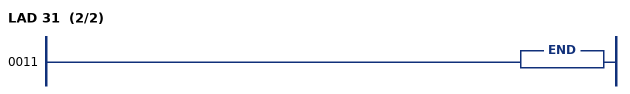
% Rung: 11 %
SOR END EOR

LADDER 32
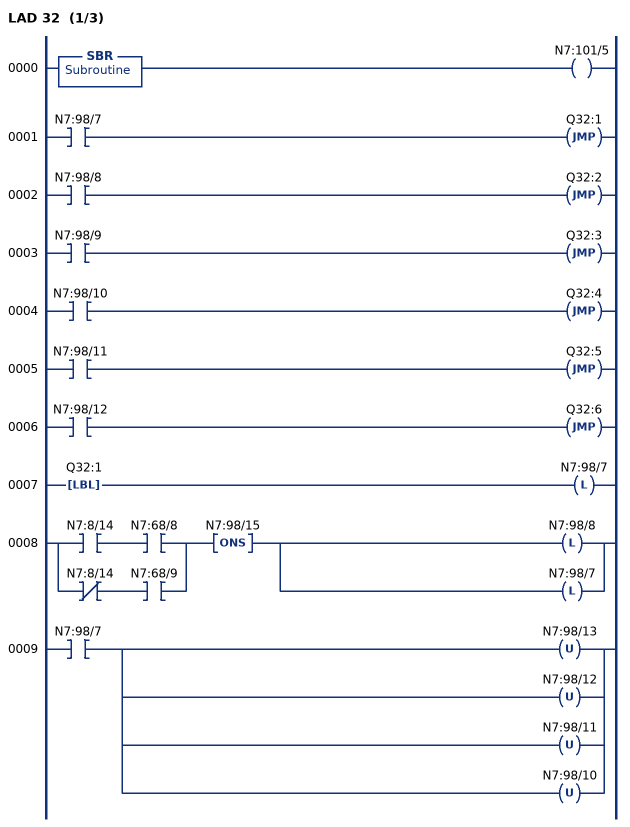
% Rung: 0 %
SOR SBR OTE N7:101/5 EOR
% Rung: 1 %
SOR XIC N7:98/7 JMP Q32:1 EOR
% Rung: 2 %
SOR XIC N7:98/8 JMP Q32:2 EOR
% Rung: 3 %
SOR XIC N7:98/9 JMP Q32:3 EOR
% Rung: 4 %
SOR XIC N7:98/10 JMP Q32:4 EOR
% Rung: 5 %
SOR XIC N7:98/11 JMP Q32:5 EOR
% Rung: 6 %
SOR XIC N7:98/12 JMP Q32:6 EOR
% Rung: 7 %
SOR LBL Q32:1 OTL N7:98/7 EOR
% Rung: 8 %
SOR BST XIC N7:8/14 XIC N7:68/8 NXB XIO N7:8/14 XIC N7:68/9 BND OSR N7:98/15 BST OTL N7:98/8 NXB OTL N7:98/7 BND EOR
% Rung: 9 %
SOR XIC N7:98/7 BST OTU N7:98/13 NXB BST OTU N7:98/12 NXB BST OTU N7:98/11 NXB OTU N7:98/10 BND BND BND EOR

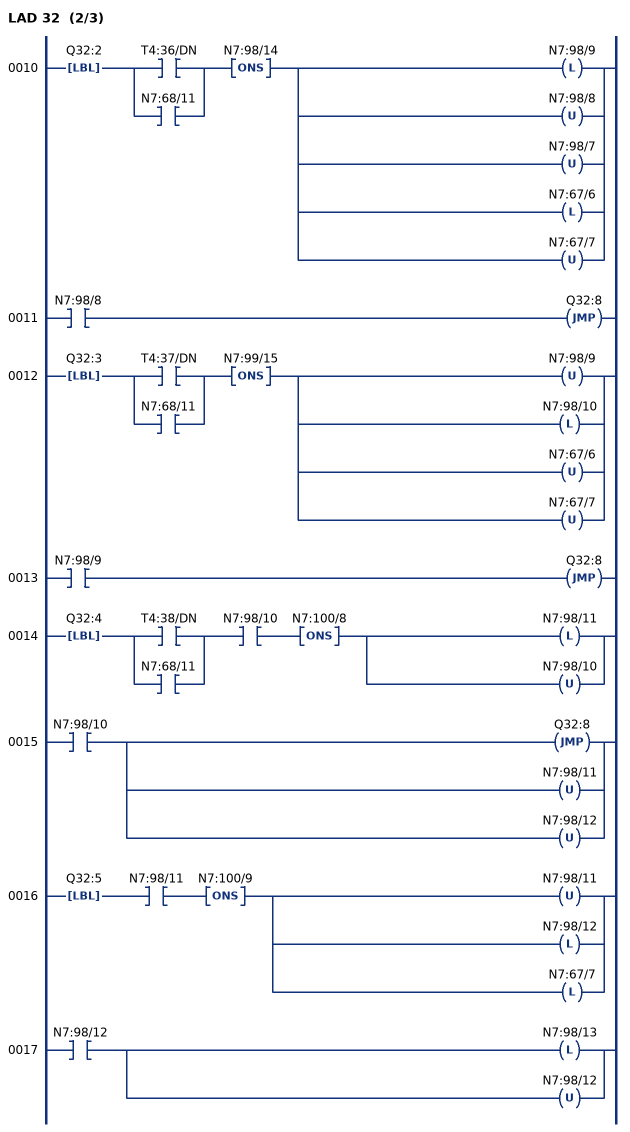
% Rung: 10 %
SOR LBL Q32:2 BST XIC T4:36/DN NXB XIC N7:68/11 BND OSR N7:98/14 BST OTL N7:98/9 NXB BST BST OTU N7:98/8 NXB OTU N7:98/7 BND NXB BST OTL N7:67/6 NXB OTU N7:67/7 BND BND BND EOR
% Rung: 11 %
SOR XIC N7:98/8 JMP Q32:8 EOR
% Rung: 12 %
SOR LBL Q32:3 BST XIC T4:37/DN NXB XIC N7:68/11 BND OSR N7:99/15 BST OTU N7:98/9 NXB BST OTL N7:98/10 NXB BST OTU N7:67/6 NXB OTU N7:67/7 BND BND BND EOR
% Rung: 13 %
SOR XIC N7:98/9 JMP Q32:8 EOR
% Rung: 14 %
SOR LBL Q32:4 BST XIC T4:38/DN NXB XIC N7:68/11 BND XIC N7:98/10 OSR N7:100/8 BST OTL N7:98/11 NXB OTU N7:98/10 BND EOR
% Rung: 15 %
SOR XIC N7:98/10 BST JMP Q32:8 NXB BST OTU N7:98/11 NXB OTU N7:98/12 BND BND EOR
% Rung: 16 %
SOR LBL Q32:5 XIC N7:98/11 OSR N7:100/9 BST BST OTU N7:98/11 NXB OTL N7:98/12 BND NXB OTL N7:67/7 BND EOR
% Rung: 17 %
SOR XIC N7:98/12 BST OTL N7:98/13 NXB OTU N7:98/12 BND EOR

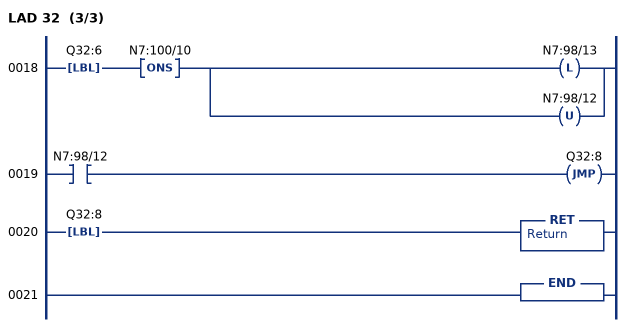
% Rung: 18 %
SOR LBL Q32:6 OSR N7:100/10 BST OTL N7:98/13 NXB OTU N7:98/12 BND EOR
% Rung: 19 %
SOR XIC N7:98/12 JMP Q32:8 EOR
% Rung: 20 %
SOR LBL Q32:8 RET EOR
% Rung: 21 %
SOR END EOR

LADDER 33
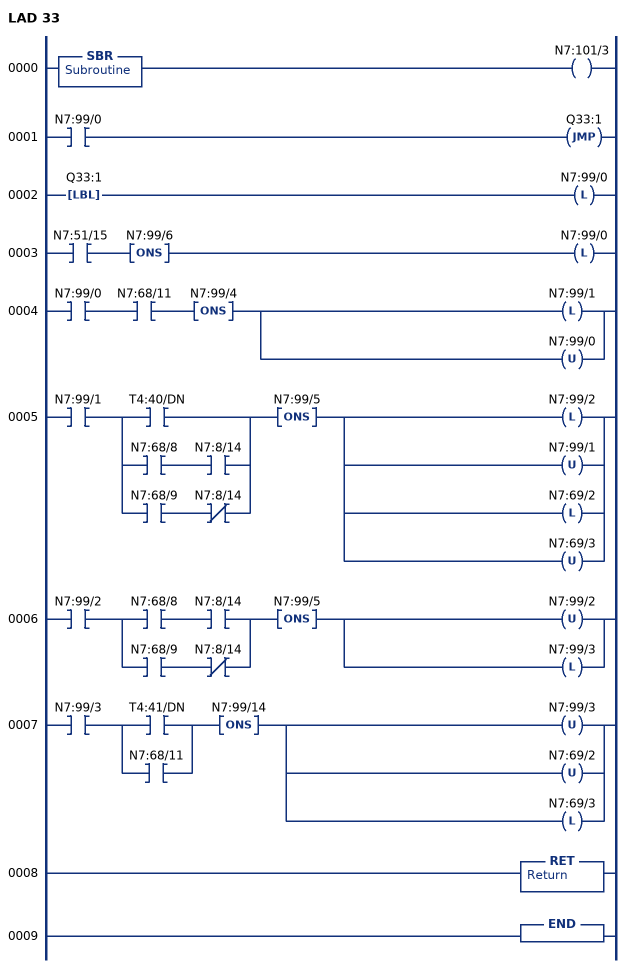
% Rung: 0 %
SOR SBR OTE N7:101/3 EOR
% Rung: 1 %
SOR XIC N7:99/0 JMP Q33:1 EOR
% Rung: 2 %
SOR LBL Q33:1 OTL N7:99/0 EOR
% Rung: 3 %
SOR XIC N7:51/15 OSR N7:99/6 OTL N7:99/0 EOR
% Rung: 4 %
SOR XIC N7:99/0 XIC N7:68/11 OSR N7:99/4 BST OTL N7:99/1 NXB OTU N7:99/0 BND EOR
% Rung: 5 %
SOR XIC N7:99/1 BST XIC T4:40/DN NXB BST XIC N7:68/8 XIC N7:8/14 NXB XIC N7:68/9 XIO N7:8/14 BND BND OSR N7:99/5 BST OTL N7:99/2 NXB BST OTU N7:99/1 NXB BST OTL N7:69/2 NXB OTU N7:69/3 BND BND BND EOR
% Rung: 6 %
SOR XIC N7:99/2 BST XIC N7:68/8 XIC N7:8/14 NXB XIC N7:68/9 XIO N7:8/14 BND OSR N7:99/5 BST OTU N7:99/2 NXB OTL N7:99/3 BND EOR
% Rung: 7 %
SOR XIC N7:99/3 BST XIC T4:41/DN NXB XIC N7:68/11 BND OSR N7:99/14 BST OTU N7:99/3 NXB BST OTU N7:69/2 NXB OTL N7:69/3 BND BND EOR
% Rung: 8 %
SOR RET EOR
% Rung: 9 %
SOR END EOR

LADDER 34
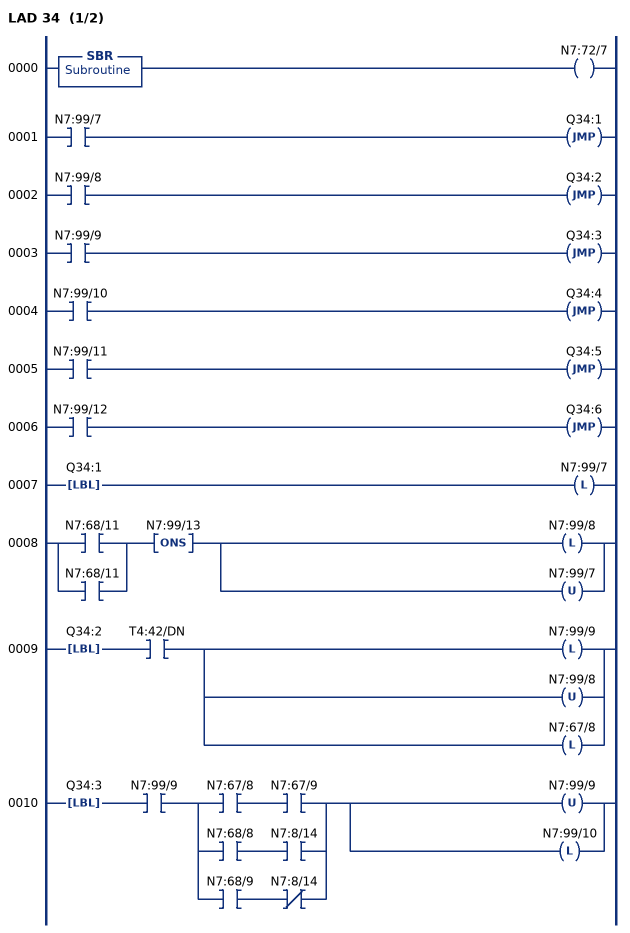
% Rung: 0 %
SOR SBR OTE N7:72/7 EOR
% Rung: 1 %
SOR XIC N7:99/7 JMP Q34:1 EOR
% Rung: 2 %
SOR XIC N7:99/8 JMP Q34:2 EOR
% Rung: 3 %
SOR XIC N7:99/9 JMP Q34:3 EOR
% Rung: 4 %
SOR XIC N7:99/10 JMP Q34:4 EOR
% Rung: 5 %
SOR XIC N7:99/11 JMP Q34:5 EOR
% Rung: 6 %
SOR XIC N7:99/12 JMP Q34:6 EOR
% Rung: 7 %
SOR LBL Q34:1 OTL N7:99/7 EOR
% Rung: 8 %
SOR BST XIC N7:68/11 NXB XIC N7:68/11 BND OSR N7:99/13 BST OTL N7:99/8 NXB OTU N7:99/7 BND EOR
% Rung: 9 %
SOR LBL Q34:2 XIC T4:42/DN BST OTL N7:99/9 NXB BST OTU N7:99/8 NXB OTL N7:67/8 BND BND EOR
% Rung: 10 %
SOR LBL Q34:3 XIC N7:99/9 BST XIC N7:67/8 XIC N7:67/9 NXB BST XIC N7:68/8 XIC N7:8/14 NXB XIC N7:68/9 XIO N7:8/14 BND BND BST OTU N7:99/9 NXB OTL N7:99/10 BND EOR

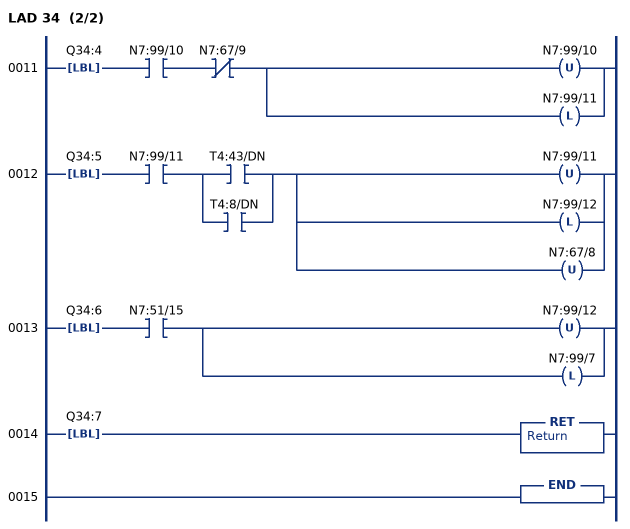
% Rung: 11 %
SOR LBL Q34:4 XIC N7:99/10 XIO N7:67/9 BST OTU N7:99/10 NXB OTL N7:99/11 BND EOR
% Rung: 12 %
SOR LBL Q34:5 XIC N7:99/11 BST XIC T4:43/DN NXB XIC T4:8/DN BND BST OTU N7:99/11 NXB BST OTL N7:99/12 NXB OTU N7:67/8 BND BND EOR
% Rung: 13 %
SOR LBL Q34:6 XIC N7:51/15 BST OTU N7:99/12 NXB OTL N7:99/7 BND EOR
% Rung: 14 %
SOR LBL Q34:7 RET EOR
% Rung: 15 %
SOR END EOR

LADDER 35
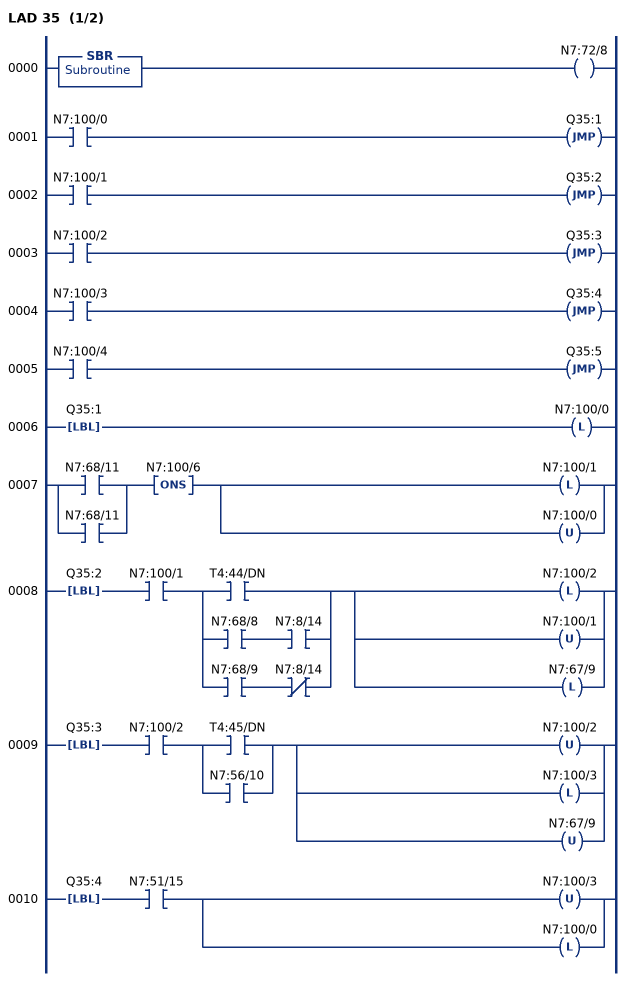
% Rung: 0 %
SOR SBR OTE N7:72/8 EOR
% Rung: 1 %
SOR XIC N7:100/0 JMP Q35:1 EOR
% Rung: 2 %
SOR XIC N7:100/1 JMP Q35:2 EOR
% Rung: 3 %
SOR XIC N7:100/2 JMP Q35:3 EOR
% Rung: 4 %
SOR XIC N7:100/3 JMP Q35:4 EOR
% Rung: 5 %
SOR XIC N7:100/4 JMP Q35:5 EOR
% Rung: 6 %
SOR LBL Q35:1 OTL N7:100/0 EOR
% Rung: 7 %
SOR BST XIC N7:68/11 NXB XIC N7:68/11 BND OSR N7:100/6 BST OTL N7:100/1 NXB OTU N7:100/0 BND EOR
% Rung: 8 %
SOR LBL Q35:2 XIC N7:100/1 BST XIC T4:44/DN NXB BST XIC N7:68/8 XIC N7:8/14 NXB XIC N7:68/9 XIO N7:8/14 BND BND BST OTL N7:100/2 NXB BST OTU N7:100/1 NXB OTL N7:67/9 BND BND EOR
% Rung: 9 %
SOR LBL Q35:3 XIC N7:100/2 BST XIC T4:45/DN NXB XIC N7:56/10 BND BST OTU N7:100/2 NXB BST OTL N7:100/3 NXB OTU N7:67/9 BND BND EOR
% Rung: 10 %
SOR LBL Q35:4 XIC N7:51/15 BST OTU N7:100/3 NXB OTL N7:100/0 BND EOR

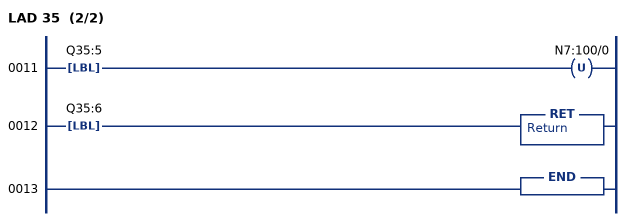
% Rung: 11 %
SOR LBL Q35:5 OTU N7:100/0 EOR
% Rung: 12 %
SOR LBL Q35:6 RET EOR
% Rung: 13 %
SOR END EOR

DATA TABLE (non-zero values as saved)
DATA T4
% .PRE .ACC %
% T4:0 % 3600 0
% T4:1 % 3800 0
% T4:2 % 3500 0
% T4:3 % 35 0
% T4:4 % 1000 0
% T4:5 % 118 0
% T4:6 % 60 0
% T4:7 % 3050 0
% T4:8 % 680 0
% T4:9 % 80 0
% T4:10 % 400 0
% T4:11 % 5 0
% T4:12 % 20 0
% T4:13 % 300 0
% T4:14 % 400 0
% T4:15 % 60 0
% T4:16 % 40 40
% T4:17 % 40 1
% T4:23 % 2000 0
% T4:24 % 500 500
% T4:25 % 10 0
% T4:26 % 2000 0
% T4:27 % 50 50
% T4:28 % 500 0
% T4:29 % 0 1
% T4:31 % 0 1
% T4:32 % 40 0
% T4:33 % 500 0
% T4:34 % 50 0
% T4:35 % 500 0
% T4:36 % 50 0
% T4:37 % 100 0
% T4:39 % 50 50
% T4:40 % 71 0
% T4:46 % 750 0
% T4:47 % 1 0
% T4:48 % 100 0
% T4:49 % 1800 0
% T4:50 % 10 0
DATA C5
% .PRE .ACC %
% C5:0 % 30000 3742
% C5:1 % 0 31359
% C5:2 % 30000 0
% C5:3 % 10 0
% C5:4 % 1000 38
DATA N7
% N7:0 % 0 0 0 0 0 0 0 0 256 3600
% N7:10 % 3800 3500 35 1000 118 60 3050 680 80 200
% N7:20 % 5 20 300 300 60 40 40 0 0 0
% N7:30 % 0 0 1700 500 10 500 50 400 0 0
% N7:40 % 0 0 0 0 -16384 0 0 0 0 0
% N7:50 % 1024 0 0 0 0 4224 1 16385 256 64
% N7:60 % 0 -32768 0 0 0 0 0 0 0 0
% N7:70 % 17328 1 0 0 0 0 16387 40 500 50
% N7:80 % 500 50 100 0 50 71 0 0 0 0
% N7:90 % 0 750 0 0 0 1 0 1152 0 0
% N7:100 % 8192 1 100 1800 10 0 0 0 0 0
DATA N10
% N10:0 % 5000 500 4300 200 4000 200 20 4500 400 20
% N10:10 % 200 20 20 150 300 50 200 400 600 800
% N10:30 % 1500 1500 1350 100 900 350 20 1300 100 100
% N10:40 % 200 20 20 150 300 50 0 200 750 950
% N10:50 % 1800 1850 1900 1900 1900 1900 1850 1850 0 380
% N10:60 % 1500 1500 1350 200 900 350 20 1300 100 20
% N10:70 % 200 20 20 110 300 50 200 400 600 800
% N10:90 % 1500 500 100 300 900 200 20 1300 150 20
% N10:100 % 200 20 20 150 300 50 200 400 600 800
% N10:120 % 1500 500 100 300 900 200 20 1300 150 20
% N10:130 % 200 20 20 150 300 50 200 400 600 800
% N10:150 % 1500 500 100 300 900 200 20 1300 150 20
% N10:160 % 200 20 20 150 300 50 200 400 600 800
% N10:180 % 1500 500 100 300 900 200 20 1300 150 20
% N10:190 % 200 20 20 150 300 50 200 400 600 800
% N10:210 % 1500 500 100 300 900 200 20 1300 150 20
% N10:220 % 200 20 20 150 300 50 200 400 600 800
% N10:250 % 2 2 1 2 1 0
